Staubli VAL3: start.pgx

program start()
  local string tt[8]
  local num l_nError
begin

  call init(l_nError)

  if l_nError<0

    popUpMsg(sErrorMessage)

  endIf

  //call _str2Array("A;   ; NON",";",tt)

end
